// TwinCAT 3 PLC project plc
// ProgramVersion: 3.1.4024.0
// libraries:
//   Tc2_Standard, * (Beckhoff Automation GmbH)
//   Tc2_System, * (Beckhoff Automation GmbH)
//   Tc3_Module, * (Beckhoff Automation GmbH)
// project tree:
//   GVLs/ InputOutput.TcGVL
//   / PlcTask.TcTTO
//   POUs/ FBAutoritenuta.TcPOU, MAIN.TcPOU
// real-time tasks:
//   TASK PlcTask: cycle T#10ms, priority 20, ADS port 350

CONFIGURATION plc
    RESOURCE PLC ON TwinCAT3
        TASK PlcTask(INTERVAL := T#10ms, PRIORITY := 20);
        PROGRAM MAIN WITH PlcTask : MAIN;
    END_RESOURCE
END_CONFIGURATION

// ---- GVLs/InputOutput.TcGVL
{attribute 'qualified_only'}
VAR_GLOBAL
	// prima macchina
	pStart	:	BOOL;
	pStop	:	BOOL;
	H1		:	BOOL;
	// seconda macchina
	pStart2	:	BOOL;
	pStop2	:	BOOL;
	H2		:	BOOL;
END_VAR

// ---- POUs/MAIN.TcPOU
PROGRAM MAIN
VAR
	Autoritenuta1: FBAutoritenuta;
	Autoritenuta2: FBAutoritenuta;
END_VAR

// prima istanza della auto ritenuta (MSF n.1)
Autoritenuta1(start:= InputOutput.pStart, stop:= InputOutput.pStop, Q => InputOutput.H1);

// seconda istanza della auto ritenuta (MSF n.2)
Autoritenuta2(start:= InputOutput.pStart2, stop:= InputOutput.pStop2 , Q => InputOutput.H2);

END_PROGRAM

// ---- POUs/FBAutoritenuta.TcPOU
FUNCTION_BLOCK FBAutoritenuta
VAR_INPUT
	start	:	BOOL;
	stop	:	BOOL;
END_VAR
VAR_OUTPUT
	Q		:	BOOL;
	Q2		:   BOOL;
END_VAR
// dichiarare le variabili di stato SOLO nella sezione VAR
VAR
	stato	:	BOOL := FALSE;
END_VAR

// IMPORTANTE:
// le variabili nel'area VAR_STAT
// sono condivise tra tutte le istanza della classe FBAutoritenuta
//  quindi:
// NON usare l'area VAR_STAT per la variabile di stato di una MSF
// altrimenti tutte le istanze della MSF si troveranno erroneamente
// nello stesso stato
//
// Invece, dichiarare le variabili di stato nell'area VAR
VAR_STAT
	statica	: BOOL;
END_VAR

// Auto ritenuta:

// 2. solo espressioni logiche
stato := (start OR stato) AND stop;

// copio la variabile di stato sull'uscita Q
Q := stato;

// copio il valore della variabile stato in statica
statica := stato;

// comando Q2 col valore della variabile statica
Q2 := statica;

END_FUNCTION_BLOCK
